(* IEC 61131-3 sources: Mirroring_Webvisu/graph/db, 7 files *)

(* ---- GRAPH_AXIS.ST ---- *)
TYPE GRAPH_AXIS :
STRUCT
	sLabel: STRING;
	aData: ARRAY[0..172803] OF REAL;
    diNumOfData : DINT;
	sBorderColor : STRING;
	xFill : BOOL;
END_STRUCT
END_TYPE

(* ---- FB_ReadTrend.ST ---- *)
FUNCTION_BLOCK FB_ReadTrend
VAR_INPUT
    xExecute : BOOL;
    sTrendName : STRING;
    tStartTime : DT;
    tEndTime : DT;
    iChannelIndex : INT := 0;
END_VAR
VAR_IN_OUT
    stChartData : GRAPH_AXIS;
END_VAR
VAR_OUTPUT
    sLabels : STRING(2000);
    xDone : BOOL;
    xBusy : BOOL;
    xError : BOOL;
    sError : STRING;
END_VAR
VAR
    step : INT := 0;
    fbTrendReader : VisuTrendStorageAccess.TrendStorageReader;
    fbTrendConsumer : FB_TrendConsumer;

    liStart : LINT;
    liEnd : LINT;
    eResult : VisuTrendStorageAccess.ETrendStorageReaderErrors;
END_VAR

CASE step OF
    0: (* Idle *)
        IF xExecute THEN
            xBusy := TRUE;
            xDone := FALSE;
            xError := FALSE;
            sError := '';

            // Set up Consumer
            fbTrendConsumer.SetDestination(ADR(stChartData), ADR(sLabels), tStartTime);

            // Initialize Reader
            fbTrendReader.Initialize(sTrendName); // User docu says Initialize exists. Assuming sTrendName arg.

            // Convert DT to LINT (Timestamp). DT is seconds. Trend usually ms.
            liStart := DT_TO_LINT(tStartTime) * 1000;
            liEnd := DT_TO_LINT(tEndTime) * 1000;

            step := 10;
        END_IF

    10: (* Start Read *)
        eResult := fbTrendReader.Read(
            liTimstampFrom := liStart,
            liTimstampTo := liEnd,
            itfTrendStorageReaderConsumer := fbTrendConsumer
        );

        IF eResult = VisuTrendStorageAccess.ETrendStorageReaderErrors.NoError THEN
             // Done immediately (unlikely for large data but possible)
             stChartData.sLabel := "Trend Data";
             stChartData.sBorderColor := "blue";
             stChartData.xFill := FALSE;
             step := 20;
        ELSIF eResult = VisuTrendStorageAccess.ETrendStorageReaderErrors.AdditionalReadCallRequired THEN
             step := 11; // Continue Reading
        ELSIF eResult = VisuTrendStorageAccess.ETrendStorageReaderErrors.NotInitialized THEN
             sError := "Not Initialized";
             xError := TRUE;
             step := 99;
        ELSE
             sError := "Read Error";
             xError := TRUE;
             step := 99;
        END_IF

    11: (* Continue Reading *)
        eResult := fbTrendReader.ContinueReading(
            liTimstampFrom := liStart,
            liTimstampTo := liEnd,
            itfTrendStorageReaderConsumer := fbTrendConsumer
        );
         IF eResult = VisuTrendStorageAccess.ETrendStorageReaderErrors.NoError THEN
             step := 20;
         ELSIF eResult = VisuTrendStorageAccess.ETrendStorageReaderErrors.AdditionalReadCallRequired THEN
             // Stay in step 11
         ELSE
             sError := "Continue Error";
             xError := TRUE;
             step := 99;
         END_IF

    20: (* Done *)
        xDone := TRUE;
        xBusy := FALSE;
        IF NOT xExecute THEN
            step := 0;
        END_IF

    99: (* Error *)
        xBusy := FALSE;
        IF NOT xExecute THEN
            step := 0;
        END_IF

END_CASE

(* ---- FB_TrendConsumer.ST ---- *)
(* Consumer FB to receive data from TrendStorageReader *)
FUNCTION_BLOCK FB_TrendConsumer IMPLEMENTS VisuTrendStorageAccess.ITrendStorageReaderConsumer
VAR
    pAxis : POINTER TO GRAPH_AXIS;
    pLabels : POINTER TO STRING(2000);
    sLabels : STRING(2000); // Internal build buffer
    iMaxLabels : INT := 20;
    tStartTime : DT;
    iCurrentRow : DINT;
    rCurrentVal : REAL;
    xFirst : BOOL := TRUE;
END_VAR

METHOD SetDestination
VAR_INPUT
    pChartData : POINTER TO GRAPH_AXIS;
    pLabelString : POINTER TO STRING(2000);
    tStart : DT;
END_VAR
    pAxis := pChartData;
    pLabels := pLabelString;
    tStartTime := tStart;

    // Reset
    IF pAxis <> 0 THEN
        pAxis^.diNumOfData := 0;
    END_IF
    IF pLabels <> 0 THEN
        pLabels^ := '[';
        sLabels := '[';
    END_IF
    xFirst := TRUE;

METHOD ErrorOccurred
VAR_INPUT
	(* The error, that occurred*)
	eETrendStorageReaderErrors	: VisuTrendStorageAccess.ETrendStorageReaderErrors;
	(* Identifies the step, where the error occurred	*)
	eDuringWhichStep	: VisuTrendStorageAccess.ETrendStorageReaderStep;
END_VAR
    // Handled in main

METHOD ReadingDataCompleted
    // Finalize labels
    IF pLabels <> 0 THEN
        pLabels^ := CONCAT(pLabels^, ']');
    END_IF

METHOD TimestampRead
VAR_INPUT
	liTimestamp	: LINT;
END_VAR
VAR
    sTempLabel : STRING(20);
    dtCurrent : DT;
    diIndex : DINT;
END_VAR
    // Convert timestamp (uS or mS? Usually uS or mS from Trend. LINT is usually ms or us)
    // Assuming MS since 1970? Or LTIME?
    // Standard Trend timestamps are µs (microseconds) usually.
    // DT is Seconds.

    // For label generation:
    IF pAxis <> 0 AND pLabels <> 0 THEN
        diIndex := pAxis^.diNumOfData; // Current index we are about to fill (ValueRead comes next usually?)
        // Actually ValueRead might come before or after? Or multiple ValueReads per timestamp.
        // Usually TimestampRead comes once per row.

        // Let's assume one variable per row for now or check iWhichVariable in ValueRead.

        IF diIndex < 100 AND (diIndex < iMaxLabels) THEN
             // Convert to DT approx
             dtCurrent := TO_DT(liTimestamp / 1000); // if ms

             sTempLabel := DT_TO_STRING(dtCurrent);
             sTempLabel := RIGHT(sTempLabel, 8);

             IF NOT xFirst THEN
                 pLabels^ := CONCAT(pLabels^, ', "');
             ELSE
                 pLabels^ := CONCAT(pLabels^, '"');
                 xFirst := FALSE;
             END_IF
             pLabels^ := CONCAT(pLabels^, sTempLabel);
             pLabels^ := CONCAT(pLabels^, '"');
        END_IF
    END_IF

METHOD ValueRead
VAR_INPUT
	diWhichRow	: DINT;
	iWhichVariable	: INT;
	liValue	: LINT;
	xValueNULL	: BOOL;
END_VAR
VAR
    diIndex : DINT;
END_VAR
    IF pAxis <> 0 THEN
        diIndex := pAxis^.diNumOfData;

        IF diIndex <= 172803 THEN
             // Convert LINT raw value to REAL.
             // Note: Raw value in Trend is often scaled. LINT might be the raw int.
             // If variable is REAL in PLC, it is stored as bit pattern or scaled???
             // Standard Trend Storage often stores as LREAL or scaled INT.
             // ValueRead signature says liValue : LINT.
             // If original var is REAL, treat LINT as bits? Or Cast?
             // For now assume direct cast or small scaling.
             pAxis^.aData[diIndex] := TO_REAL(liValue);

             pAxis^.diNumOfData := pAxis^.diNumOfData + 1;
        END_IF
    END_IF

METHOD VariableConfigurationRead
VAR_INPUT
	pVariableConfiguration	: POINTER TO VisuTrendStorageAccess.TblTrendVariable;
	xIsFirstVariableConfiguration	: BOOL;
END_VAR
    // Optional
END_FUNCTION_BLOCK

(* ---- read_db.ST ---- *)
TYPE GRAPH_AXIS :
STRUCT
	sLabel: STRING;
	aData: ARRAY[0..172803] OF REAL;
    diNumOfData : DINT;
	sBorderColor : STRING;
	xFill : BOOL;
END_STRUCT
END_TYPE

(* Consumer FB to receive data from TrendStorageReader *)
FUNCTION_BLOCK FB_TrendConsumer IMPLEMENTS VisuTrendStorageAccess.ITrendStorageReaderConsumer
VAR
    pAxis : POINTER TO GRAPH_AXIS;
    pLabels : POINTER TO STRING(2000);
    sLabels : STRING(2000); // Internal build buffer
    iMaxLabels : INT := 20;
    tStartTime : DT;
    iCurrentRow : DINT;
    rCurrentVal : REAL;
    xFirst : BOOL := TRUE;
END_VAR

METHOD SetDestination
VAR_INPUT
    pChartData : POINTER TO GRAPH_AXIS;
    pLabelString : POINTER TO STRING(2000);
    tStart : DT;
END_VAR
    pAxis := pChartData;
    pLabels := pLabelString;
    tStartTime := tStart;

    // Reset
    IF pAxis <> 0 THEN
        pAxis^.diNumOfData := 0;
    END_IF
    IF pLabels <> 0 THEN
        pLabels^ := '[';
        sLabels := '[';
    END_IF
    xFirst := TRUE;

METHOD ErrorOccurred
VAR_INPUT
	eErrorCode	: VisuTrendStorageAccess.ETrendStorageReaderErrors;
END_VAR
    // Handled in main

METHOD ReadingDataCompleted
    // Finalize labels
    IF pLabels <> 0 THEN
        pLabels^ := CONCAT(pLabels^, ']');
    END_IF

METHOD TimestampRead
VAR_INPUT
	liTimestamp	: LINT;
END_VAR
VAR
    sTempLabel : STRING(20);
    dtCurrent : DT;
    diIndex : DINT;
END_VAR
    // Convert timestamp (uS or mS? Usually uS or mS from Trend. LINT is usually ms or us)
    // Assuming MS since 1970? Or LTIME?
    // Standard Trend timestamps are µs (microseconds) usually.
    // DT is Seconds.

    // For label generation:
    IF pAxis <> 0 AND pLabels <> 0 THEN
        diIndex := pAxis^.diNumOfData; // Current index we are about to fill (ValueRead comes next usually?)
        // Actually ValueRead might come before or after? Or multiple ValueReads per timestamp.
        // Usually TimestampRead comes once per row.

        // Let's assume one variable per row for now or check iWhichVariable in ValueRead.

        IF diIndex < 100 AND (diIndex < iMaxLabels) THEN
             // Convert to DT approx
             dtCurrent := TO_DT(liTimestamp / 1000); // if ms

             sTempLabel := DT_TO_STRING(dtCurrent);
             sTempLabel := RIGHT(sTempLabel, 8);

             IF NOT xFirst THEN
                 pLabels^ := CONCAT(pLabels^, ', "');
             ELSE
                 pLabels^ := CONCAT(pLabels^, '"');
                 xFirst := FALSE;
             END_IF
             pLabels^ := CONCAT(pLabels^, sTempLabel);
             pLabels^ := CONCAT(pLabels^, '"');
        END_IF
    END_IF

METHOD ValueRead
VAR_INPUT
	diWhichRow	: DINT;
	iWhichVariable	: INT;
	liValue	: LINT;
	xValueNULL	: BOOL;
END_VAR
VAR
    diIndex : DINT;
END_VAR
    IF pAxis <> 0 THEN
        diIndex := pAxis^.diNumOfData;

        IF diIndex <= 172803 THEN
             // Convert LINT raw value to REAL.
             // Note: Raw value in Trend is often scaled. LINT might be the raw int.
             // If variable is REAL in PLC, it is stored as bit pattern or scaled???
             // Standard Trend Storage often stores as LREAL or scaled INT.
             // ValueRead signature says liValue : LINT.
             // If original var is REAL, treat LINT as bits? Or Cast?
             // For now assume direct cast or small scaling.
             pAxis^.aData[diIndex] := TO_REAL(liValue);

             pAxis^.diNumOfData := pAxis^.diNumOfData + 1;
        END_IF
    END_IF

METHOD VariableConfigurationRead
VAR_INPUT
	pVariableConfiguration	: POINTER TO VisuTrendStorageAccess.TblTrendVariable;
	xIsFirstVariableConfiguration	: BOOL;
END_VAR
    // Optional
END_FUNCTION_BLOCK

FUNCTION_BLOCK FB_ReadTrend
VAR_INPUT
    xExecute : BOOL;
    sTrendName : STRING;
    tStartTime : DT;
    tEndTime : DT;
    iChannelIndex : INT := 0;
END_VAR
VAR_IN_OUT
    stChartData : GRAPH_AXIS;
END_VAR
VAR_OUTPUT
    sLabels : STRING(2000);
    xDone : BOOL;
    xBusy : BOOL;
    xError : BOOL;
    sError : STRING;
END_VAR
VAR
    step : INT := 0;
    fbTrendReader : VisuTrendStorageAccess.TrendStorageReader;
    fbTrendConsumer : FB_TrendConsumer;

    liStart : LINT;
    liEnd : LINT;
    eResult : VisuTrendStorageAccess.ETrendStorageReaderErrors;
END_VAR

CASE step OF
    0: (* Idle *)
        IF xExecute THEN
            xBusy := TRUE;
            xDone := FALSE;
            xError := FALSE;
            sError := '';

            // Set up Consumer
            fbTrendConsumer.SetDestination(ADR(stChartData), ADR(sLabels), tStartTime);

            // Initialize Reader
            fbTrendReader.Initialize(sTrendName); // User docu says Initialize exists. Assuming sTrendName arg.

            // Convert DT to LINT (Timestamp). DT is seconds. Trend usually ms.
            liStart := DT_TO_LINT(tStartTime) * 1000;
            liEnd := DT_TO_LINT(tEndTime) * 1000;

            step := 10;
        END_IF

    10: (* Start Read *)
        eResult := fbTrendReader.Read(
            liTimstampFrom := liStart,
            liTimstampTo := liEnd,
            itfTrendStorageReaderConsumer := fbTrendConsumer
        );

        IF eResult = VisuTrendStorageAccess.ETrendStorageReaderErrors.NoError THEN
             // Done immediately (unlikely for large data but possible)
             stChartData.sLabel := "Trend Data";
             stChartData.sBorderColor := "blue";
             stChartData.xFill := FALSE;
             step := 20;
        ELSIF eResult = VisuTrendStorageAccess.ETrendStorageReaderErrors.AdditionalReadCallRequired THEN
             step := 11; // Continue Reading
        ELSIF eResult = VisuTrendStorageAccess.ETrendStorageReaderErrors.NotInitialized THEN
             sError := "Not Initialized";
             xError := TRUE;
             step := 99;
        ELSE
             sError := "Read Error";
             xError := TRUE;
             step := 99;
        END_IF

    11: (* Continue Reading *)
        eResult := fbTrendReader.ContinueReading(
            itfTrendStorageReaderConsumer := fbTrendConsumer
        );
         IF eResult = VisuTrendStorageAccess.ETrendStorageReaderErrors.NoError THEN
             step := 20;
         ELSIF eResult = VisuTrendStorageAccess.ETrendStorageReaderErrors.AdditionalReadCallRequired THEN
             // Stay in step 11
         ELSE
             sError := "Continue Error";
             xError := TRUE;
             step := 99;
         END_IF

    20: (* Done *)
        xDone := TRUE;
        xBusy := FALSE;
        IF NOT xExecute THEN
            step := 0;
        END_IF

    99: (* Error *)
        xBusy := FALSE;
        IF NOT xExecute THEN
            step := 0;
        END_IF

END_CASE

(* ---- PRG_TrendReadExample.ST ---- *)
PROGRAM PRG_TrendReadExample
VAR
    (* Function Block Instance *)
    fbTrendReader : FB_ReadTrend;

    (* Data Structure for the Chart *)
    stMyChartData : GRAPH_AXIS;
    sMyLabels : STRING(2000);

    (* Control Variables *)
    xReadTrigger : BOOL;
    xDone : BOOL;
    xBusy : BOOL;
    xError : BOOL;
    sErrorMessage : STRING;

    (* Parameters *)
    dtStartTime : DT;
    dtEndTime : DT;
    sTrendName : STRING := 'Trend1'; (* MUST match the Trend Recording name in Visualization Manager *)

    (* Helper to calc times *)
    tDuration : TIME := T#1H; (* Read last 1 hour *)
    // fbGetTime : GetLocalTime; (* Placeholder: Use system specific time FB *)
    dtNow : DT := DT#2024-01-01-10:00:00; (* Replace with actual system time *)
END_VAR

(*
    Example Usage:
    1. Set 'xReadTrigger' to TRUE to start reading.
    2. The FB will fetch data from 'Trend1' for the specified time range.
    3. 'stMyChartData' and 'sMyLabels' will be populated.
    4. Link 'stMyChartData' and 'sMyLabels' to your WebVisu Chart.
*)

IF xReadTrigger AND NOT xBusy THEN
    (* 1. Setup Time Range (Example: Last 1 Hour) *)
    // dtNow := ... (Get System Time here)
    dtEndTime := dtNow;
    dtStartTime := dtNow - tDuration;

    (* 2. Reset Status *)
    xReadTrigger := FALSE; (* Auto-reset trigger *)

    (* 3. Call FB *)
    fbTrendReader(
        xExecute := TRUE,
        sTrendName := sTrendName,
        tStartTime := dtStartTime,
        tEndTime := dtEndTime,
        stChartData := stMyChartData
    );
ELSE
    (* Cyclic Call *)
    fbTrendReader(
        xExecute := FALSE, (* Only TRUE for one cycle to start, or hold TRUE until Done? Implementation depends on FB logic *)
        (* Note: In the FB implementation, xExecute acts as a rising edge trigger for step 0->10 *)
        stChartData := stMyChartData
    );
END_IF

(* Output Mapping *)
sMyLabels := fbTrendReader.sLabels;
xDone := fbTrendReader.xDone;
xBusy := fbTrendReader.xBusy;
xError := fbTrendReader.xError;
sErrorMessage := fbTrendReader.sError;

(*
   Visualization Linkage:
   - Pass 'stMyChartData' components (sLabel, aData, sBorderColor, xFill) to the Chart properties.
   - Pass 'sMyLabels' to the Chart's 'InputLabels' property.
*)

(* ---- read_trend.ST ---- *)
PROGRAM read_trend
VAR
    (* Function Block Instance *)
    fbTrendReader : FB_ReadTrend;

    (* Data Structure for the Chart *)
    stMyChartData : GRAPH_AXIS;
    sMyLabels : STRING(2000);

    (* Control Variables *)
    xReadTrigger : BOOL;
    xDone : BOOL;
    xBusy : BOOL;
    xError : BOOL;
    sErrorMessage : STRING;

    (* Parameters *)
    dtStartTime : DT;
    dtEndTime : DT;
    sTrendName : STRING := 'Trend1'; (* MUST match the Trend Recording name *)

    (* Helper to calc times *)
    tDuration : TIME := T#1H; (* Read last 1 hour to ensure we get at least 100 points *)
    dtNow : DT;

    (* Time Helper *)
    stUTC_DateAndTime : SysTimeRtc.SYSTIME;
    ldtNow : LDATE_AND_TIME;
    udiResult : RTS_IEC_RESULT;

    (* Post-processing *)
    i : DINT;
    diOffset : DINT;
END_VAR

// Cyclic Call to update time
udiResult := SysTimeRtc.SysTimeRtcHighResGet(stUTC_DateAndTime);
ldtNow := TO_LDT(stUTC_DateAndTime * LTIME#1ms);
dtNow := TO_DT(ldtNow);

IF xReadTrigger AND NOT xBusy THEN
    (* 1. Setup Time Range *)
    dtEndTime := dtNow;

    // Prevent underflow
    IF dtNow > TO_DT(TIME_TO_DWORD(tDuration)) THEN
        dtStartTime := dtNow - tDuration;
    ELSE
        dtStartTime := DT#1970-01-01-00:00:00;
    END_IF

    (* 2. Reset Status *)
    xReadTrigger := FALSE;

    (* 3. Call FB *)
    fbTrendReader(
        xExecute := TRUE,
        sTrendName := sTrendName,
        tStartTime := dtStartTime,
        tEndTime := dtEndTime,
        stChartData := stMyChartData
    );
ELSE
    (* Cyclic Call *)
    fbTrendReader(
        xExecute := FALSE,
        stChartData := stMyChartData
    );
END_IF

(* Output Mapping *)
xDone := fbTrendReader.xDone;
xBusy := fbTrendReader.xBusy;
xError := fbTrendReader.xError;
sErrorMessage := fbTrendReader.sError;
sMyLabels := fbTrendReader.sLabels;

(* 4. Truncate to last 100 if needed *)
IF xDone AND NOT xError THEN
    IF stMyChartData.diNumOfData > 100 THEN
        diOffset := stMyChartData.diNumOfData - 100;

        // Shift data to the left
        FOR i := 0 TO 99 DO
            stMyChartData.aData[i] := stMyChartData.aData[i + diOffset];
        END_FOR

        // Update count
        stMyChartData.diNumOfData := 100;

        // Note: Labels are string based and harder to shift perfectly without parsing 'sLabels',
        // so we might leave them or clear them if strict alignment is needed.
        // For now, we leave them as is, but data is truncated.
    END_IF
END_IF

(* ---- test_Value.ST ---- *)
PROGRAM test_Value
VAR
    stChartData : GRAPH_AXIS;
    xInit : BOOL := TRUE;
END_VAR

(* Initialize only once or on demand *)
IF xInit THEN
    (* 1. Set Style Properties - Using fields from graph/db/GRAPH_AXIS.ST *)
    stChartData.sLabel := 'Fixed Values Demo';
    stChartData.sBorderColor := 'rgb(54, 162, 235)'; (* Blue *)
    stChartData.xFill := FALSE;

    (* 2. Set 10 Fixed Data Points *)
    stChartData.aData[0] := 10.0;
    stChartData.aData[1] := 20.0;
    stChartData.aData[2] := 15.5;
    stChartData.aData[3] := 25.0;
    stChartData.aData[4] := 30.0;
    stChartData.aData[5] := 10.0;
    stChartData.aData[6] := 5.0;
    stChartData.aData[7] := 12.0;
    stChartData.aData[8] := 18.0;
    stChartData.aData[9] := 22.0;

    (* Set the number of valid data points *)
    stChartData.diNumOfData := 10;

    xInit := FALSE;
END_IF
